(* IEC 61131-3 sources: Elmo_Master/Lasal_PRG/Elmo_EtherCAT_Test_4Axis/Class/LMCRecorderStore (part 2) *)

END_FUNCTION

FUNCTION LMCRecorderStore::LMCRecorderStore
	VAR_OUTPUT
		ret_code 	: ConfStates;
	END_VAR
	VAR
		bankIndex : UINT;
	END_VAR

	StateValue := LMC_RECORDER_EMPTY;
	ConfigId := 0;
	ConfigRevision := 0;
	MapRevision := 0;
	OwnerSessionEpoch := 0;
	ClosedSessionEpoch := 0;
	DiagnosticsBootId := 0;
	RecordId := 0;
	BufferId := 0;
	SampleCapacity := 0;
	SampleCount := 0;
	SamplePeriodCycles := 1;
	ChannelCount := 0;
	SampleStrideBytes := 0;
	BufferMode := 0;
	TriggerType := 0;
	TriggerValueType := 0;
	TriggerOperator := 0;
	PreTriggerSamples := 0;
	PostTriggerSamples := 0;
	TriggerSignalId := 0;
	TriggerSignalOffset := 0;
	TriggerValue := 0;
	TriggerMask := 0;
	CapturePhase := 1;
	StopReason := LMC_RECORDER_STOP_NONE;
	TriggerIndex := 0xFFFFFFFF;
	TriggerCycle := 0;
	TriggerTimestampLow := 0;
	TriggerTimestampHigh := 0;
	StartCycle := 0;
	EndCycle := 0;
	StartTimestampLow := 0;
	StartTimestampHigh := 0;
	EndTimestampLow := 0;
	EndTimestampHigh := 0;
	DroppedCycles := 0;
	OverflowCount := 0;
	DividerCounter := 0;
	NextConfigId := 1;
	NextRecordId := 1;
	StartRequestSequence := 0;
	StartAppliedSequence := 0;
	TriggerRequestSequence := 0;
	TriggerAppliedSequence := 0;
	StopRequestSequence := 0;
	StopAppliedSequence := 0;
	StatusSequence := 0;
	WriteSampleIndex := 0;
	FrozenFirstSampleIndex := 0;
	PostSamplesRemaining := 0;
	PreviousTriggerValue := 0;
	PreviousTriggerValid := FALSE;
	BufferReleased := TRUE;
	_memset(dest:=#SignalIds[0], usByte:=0, cntr:=sizeof(SignalIds));
	_memset(dest:=#SignalOffsets[0], usByte:=0, cntr:=sizeof(SignalOffsets));
	g_LMCRecorderRecoveryToken[0] := 0;
	g_LMCRecorderRecoveryToken[1] := 0;
	g_LMCRecorderRecoveryToken[2] := 0;
	g_LMCRecorderRecoveryToken[3] := 0;
	g_LMCRecorderLastReleasedRecoveryToken[0] := 0;
	g_LMCRecorderLastReleasedRecoveryToken[1] := 0;
	g_LMCRecorderLastReleasedRecoveryToken[2] := 0;
	g_LMCRecorderLastReleasedRecoveryToken[3] := 0;
	sigclib_atomic_setU32(
		pValue:=#g_LMCRecorderActiveGeneration, value:=0);
	for bankIndex := 0 to LMC_RECORDER_BANK_COUNT - 1 do
		g_LMCRecorderBankRecordId[bankIndex] := 0;
		g_LMCRecorderBankConfigId[bankIndex] := 0;
		g_LMCRecorderBankConfigRevision[bankIndex] := 0;
		g_LMCRecorderBankMapRevision[bankIndex] := 0;
		g_LMCRecorderBankOwnerSessionEpoch[bankIndex] := 0;
		g_LMCRecorderBankClosedSessionEpoch[bankIndex] := 0;
		g_LMCRecorderBankDiagnosticsBootId[bankIndex] := 0;
		g_LMCRecorderBankSampleCapacity[bankIndex] := 0;
		g_LMCRecorderBankSampleCount[bankIndex] := 0;
		g_LMCRecorderBankCapturePhase[bankIndex] := 0;
		g_LMCRecorderBankStopReason[bankIndex] := 0;
		g_LMCRecorderBankTriggerIndex[bankIndex] := 0xFFFFFFFF;
		g_LMCRecorderBankTriggerCycle[bankIndex] := 0;
		g_LMCRecorderBankTriggerTimestampLow[bankIndex] := 0;
		g_LMCRecorderBankTriggerTimestampHigh[bankIndex] := 0;
		g_LMCRecorderBankStartCycle[bankIndex] := 0;
		g_LMCRecorderBankEndCycle[bankIndex] := 0;
		g_LMCRecorderBankStartTimestampLow[bankIndex] := 0;
		g_LMCRecorderBankStartTimestampHigh[bankIndex] := 0;
		g_LMCRecorderBankEndTimestampLow[bankIndex] := 0;
		g_LMCRecorderBankEndTimestampHigh[bankIndex] := 0;
		g_LMCRecorderBankDroppedCycles[bankIndex] := 0;
		g_LMCRecorderBankOverflowCount[bankIndex] := 0;
		g_LMCRecorderBankFrozenFirstSampleIndex[bankIndex] := 0;
		sigclib_atomic_setU32(
			pValue:=#g_LMCRecorderBankState[bankIndex],
			value:=LMC_RECORDER_EMPTY);
	end_for;
	ret_code := C_OK;

END_FUNCTION
